TYPE ST_WarehouseBackFeeback :
STRUCT
	//提供圓帶上的針數
	AllocationInfo : ARRAY[0..40] OF st_AllocationData;
END_STRUCT
END_TYPE

(* stored: Version 1.1.0.1, ProductVersion 3.1.4024.13
   DUT ST_WarehouseBackFeeback: Id {19087237-38ac-4a80-93ab-cfdd08c6814c} *)
